(*

.. <legal notes>

legal notes
=================
| SPDX-FileCopyrightText: © 2026 Oleksandr Tiutyk <trofimich@gmail.com>
| SPDX-License-Identifier: LGPL-3.0-only
| For details check: LGPL-3.0-only_

.. _LGPL-3.0-only: https://www.gnu.org/licenses/lgpl-3.0.en.html

.. </legal notes>

*)

{attribute 'no_explicit_call' := 'do not call this POU directly'}
PROGRAM CurrentNamespace
VAR
	{attribute 'hide'} 
	_NamespaceExtractor : NamespaceExtractor;
END_VAR

{attribute 'monitoring' := 'call'}
PROPERTY Name : STRING
GET
Name := _NamespaceExtractor.CurrentNamespace;
END_GET
END_PROPERTY

END_PROGRAM

(* stored: Version 1.1.0.1
   POU CurrentNamespace: Id {29d59fb8-a159-434c-845e-25416abc76be}, SpecialFunc None
   Property Name: Id {f675da5f-d0b6-41fc-bd89-6621afb10832}
   Get Get: Id {cbb8be66-75a1-408a-8ff6-bd79cce93d2c} *)
